// TIA Portal V19 export
DATA_BLOCK "CallEquipment_DB"   // DB38
AUTHOR : Siemens_FA_SUP
// stored: InstanceOfName Unit2.EM4.CallEquipment, InstanceOfType FB, Namespace Unit2.EM4
"Unit2.EM4.CallEquipment"
   // VAR_IN_OUT
   //    unitStatus : "LAF_typeUnitStatus";
   //    unitAlarmDB : "LAF_typeAlarms";
   //    emFeedback : "LUC_typeEmFeedback";
   // END_VAR
   // VAR
   //    statUnitStatus { ExternalWritable := 'False'} : "LAF_typeUnitStatus";
   //    instJobExecute { ExternalWritable := 'False'} : "LAF_SelectJob";
   //    instJobStopping { ExternalWritable := 'False'; S7_SetPoint := 'True'} : "LAF_SelectJob";
   //    instJobStarting { ExternalWritable := 'False'; S7_SetPoint := 'True'} : "LAF_SelectJob";
   //    instJobHolding { ExternalWritable := 'False'; S7_SetPoint := 'True'} : "LAF_SelectJob";
   //    instJobUnHolding { ExternalWritable := 'False'; S7_SetPoint := 'True'} : "LAF_SelectJob";
   //    instJobRecover { ExternalWritable := 'False'; S7_SetPoint := 'True'} : "LAF_SelectJob";
   //    instJobReseting { ExternalWritable := 'False'; S7_SetPoint := 'True'} : "LAF_SelectJob";
   //    instSequence { ExternalWritable := 'False'} : "Unit2.EM4.Sequence";
   //    instManageBitAlarms { ExternalWritable := 'False'} : "LAF_ManageBitAlarms";
   //    instCmReset { ExternalWritable := 'False'} : "Unit2.EM4.EXCHANGETRAY_ConstraintRollerCmResetOperator";
   //    instCm8SignalTM { ExternalWritable := 'False'; S7_SetPoint := 'True'} : "LEXCHANGETRAY_U2Em4SingleTM";
   //    instCm1Axis { ExternalWritable := 'False'} : "LBC_AxisSimpleControl";
   //    instCm2Axis { ExternalWritable := 'False'; S7_SetPoint := 'True'} : "LBC_AxisSimpleControl";
   //    instCm3Axis { ExternalWritable := 'False'; S7_SetPoint := 'True'} : "LBC_AxisSimpleControl";
   //    instCm4Cylinder { ExternalWritable := 'False'; S7_SetPoint := 'True'} : "LEXCHANGETRAY_Cylinder";
   //    instCm5Cylinder { ExternalWritable := 'False'; S7_SetPoint := 'True'} : "LEXCHANGETRAY_Cylinder";
   //    instCm6Cylinder { ExternalWritable := 'False'; S7_SetPoint := 'True'} : "LEXCHANGETRAY_Cylinder";
   //    instCm7Cylinder { ExternalWritable := 'False'; S7_SetPoint := 'True'} : "LEXCHANGETRAY_Cylinder";
   //    statLstUnitMode { ExternalWritable := 'False'; S7_SetPoint := 'True'} : DInt;
   // END_VAR
BEGIN
END_DATA_BLOCK
